(* IEC 61131-3 sources: teller/JD_Teller_LC2_V11/Class/Jamdetection_TeachIn_Teller, 1 file *)

(* ---- Jamdetection_TeachIn_Teller.st ---- *)
(*!
<Class
	Name               = "Jamdetection_TeachIn_Teller"
	Revision           = "1.1"
	RealtimeTask       = "true"
	CyclicTask         = "true"
	BackgroundTask     = "false"
	Sigmatek           = "false"
	OSInterface        = "false"
	HighPriority       = "false"
	Automatic          = "false"
	UpdateMode         = "Prescan"
	SharedCommandTable = "true"
	Objectsize         = "(540,120)">
	<Channels>
		<Server Name="ClassSvr" Visualized="false" Initialize="false" WriteProtected="true" Retentive="false"/>
		<Server Name="CopyTeachIn" Visualized="true" Initialize="false" WriteProtected="false" Retentive="false"/>
		<Server Name="iEncDiv" Visualized="true" Initialize="false" WriteProtected="false" Retentive="false"/>
		<Server Name="iEncMulti" Visualized="true" Initialize="false" WriteProtected="false" Retentive="false"/>
		<Server Name="JamPauze" Visualized="true" Initialize="false" WriteProtected="false" Retentive="false"/>
		<Server Name="MaxLengthBox" Visualized="true" Initialize="false" WriteProtected="false" Retentive="false"/>
		<Server Name="MinJamSpeed" Visualized="true" Initialize="false" WriteProtected="false" Retentive="false"/>
		<Server Name="MinSpot" Visualized="true" Initialize="false" WriteProtected="false" Retentive="false"/>
		<Server Name="Nr_Of_JamSensors" Visualized="true" Initialize="false" WriteProtected="true" Retentive="false"/>
		<Server Name="oJamdetection" Visualized="true" Initialize="false" WriteProtected="true" Retentive="false"/>
		<Server Name="oSpeed" Visualized="true" Initialize="false" WriteProtected="true" Retentive="false"/>
		<Server Name="ResetJam" Visualized="false" Initialize="false" WriteProtected="false" Retentive="false"/>
		<Server Name="Sectie" Visualized="true" Initialize="false" WriteProtected="true" Retentive="false"/>
		<Server Name="SectieNrInMachine" Visualized="true" Initialize="false" WriteProtected="false" Retentive="false"/>
		<Server Name="SectieType" Visualized="true" Initialize="false" WriteProtected="true" Retentive="false"/>
		<Server Name="sExtraBox" Visualized="true" Initialize="false" WriteProtected="false" Retentive="false"/>
		<Server Name="SimSpeed" Visualized="false" Initialize="false" WriteProtected="false" Retentive="false"/>
		<Server Name="Simulator" Visualized="false" Initialize="false" WriteProtected="false" Retentive="false"/>
		<Server Name="TeachIn" Visualized="true" Initialize="false" WriteProtected="false" Retentive="false"/>
		<Client Name="c_JamData" Required="true" Internal="false"/>
		<Client Name="c_SectieType" Required="true" Internal="false"/>
		<Client Name="cJamDetect" Required="false" Internal="false" Comment="Status Jamdetect&#13;&#10;1: Detectie&#13;&#10;0: Geen detectie"/>
		<Client Name="cJamDetect2HW" Required="true" Internal="false"/>
		<Client Name="cJamDetectSignal" Required="false" Internal="false" Comment="Knipperende uitgang"/>
		<Client Name="cJamReset" Required="true" Internal="false"/>
		<Client Name="cSensor_01" Required="false" Internal="false"/>
		<Client Name="cSensor_02" Required="false" Internal="false"/>
		<Client Name="cSensor_03" Required="false" Internal="false"/>
		<Client Name="cSimpuls" Required="false" Internal="false"/>
		<Client Name="iEncoder" Required="false" Internal="false"/>
	</Channels>
	<RevDoku>
		<Owner Company="jd" Author="SV"/>
		<Dokumentation Revision="1.1" Date="2014-09-16" Author="SV" Company="jd" Description="Clients cSensor_4 tm cSensor_16 verwijderd.&#13;&#10;cSimpuls sensoren verwijderd.&#13;&#10;TaskOnOff server verwijderd.&#13;&#10;TaskOnOff uit RT en CY wordk verwijderd."/>
		<Dokumentation Revision="1.0" Date="2014-09-04" Author="SV" Company="jd" Description="Kopie uit retrofit class versie 1.2. De class haalt de neemt nu de EncMul, EncDiv, MinSpot en &#13;&#10;ExtraBox uit de TellerClass_Teller.&#13;&#10;Client Jampauze ingevoerd, regel 244. Zorgt voor tijdelijk negeren van de jamfunctie."/>
	</RevDoku>
</Class>
*)
Jamdetection_TeachIn_Teller : CLASS
	TYPE
#pragma pack(push, 1)
	  tJam : STRUCT
	    Sensor : ARRAY [0..16] OF DINT;
	    CaseMinSSW : ARRAY [0..16] OF DINT;
	    MinimaleCounter : ARRAY [0..16] OF DINT;
	    Din : ARRAY [0..16] OF DINT;
	    JamBoxlength : ARRAY [0..16] OF DINT;
	    JamBoxLengthCalc : ARRAY [0..16] OF DINT;
	    CaseJam : ARRAY [0..16] OF DINT;
	    Jampos : ARRAY [0..16] OF DINT;
	    Jamdetection : ARRAY [0..16] OF DINT;
	    CaseTeachIn : ARRAY [0..16] OF DINT;
	    TeachInLength : ARRAY [0..16] OF DINT;
	    Holes : ARRAY [0..16] OF DINT;
	    Sensor_Aanwezig : ARRAY [0..16] OF DINT;
	    OnOff : ARRAY [0..16] OF DINT;
	  END_STRUCT;
#pragma pack(pop)
	END_TYPE
  //Servers:
	ClassSvr 	: SvrChCmd_DINT;
	Sectie 	: SvrCh_tSectie;
	SectieType 	: SvrCh_DINT;
	Nr_Of_JamSensors 	: SvrCh_DINT;
	SectieNrInMachine 	: SvrCh_DINT;
	MinJamSpeed 	: SvrCh_DINT;
	MinSpot 	: SvrCh_DINT;
	sExtraBox 	: SvrCh_DINT;
	iEncMulti 	: SvrCh_DINT;
	iEncDiv 	: SvrCh_DINT;
	oSpeed 	: SvrCh_DINT;
	SimSpeed 	: SvrCh_DINT;
	Simulator 	: SvrCh_DINT;
	MaxLengthBox 	: SvrCh_DINT;
	oJamdetection 	: SvrCh_DINT;
	ResetJam 	: SvrCh_DINT;
	TeachIn 	: SvrCh_DINT;
	CopyTeachIn 	: SvrCh_DINT;
	JamPauze 	: SvrCh_DINT;
  //Clients:
	c_JamData 	: CltChCmd_RAMex;
	c_SectieType 	: CltCh_DINT;
	iEncoder 	: CltCh_DINT;
	cJamDetect 	: CltCh_DINT;
	cJamDetectSignal 	: CltCh_DINT;
	cJamDetect2HW 	: CltCh_DINT;
	cSensor_01 	: CltCh_DINT;
	cSensor_02 	: CltCh_DINT;
	cSensor_03 	: CltCh_DINT;
	cSimpuls 	: CltCh_DINT;
	cJamReset 	: CltCh_DINT;
  //Variables:
		JamData 	: ^tJamDetect;
		Enc 	: Encoder1;
		Jam 	: tJam;
		OSpeedie 	: tOspeed;
		i 	: DINT;
		ii 	: DINT;
		iii 	: DINT;
		Reset 	: DINT;
		Teach 	: DINT;
		Timer 	: UDINT;
		Timer2 	: UDINT;
		Timer3 	: UDINT;
		caseKnipper 	: DINT;
		cJamDetectSignalOld 	: DINT;
		caseJam2HW 	: DINT;
		JamDetPrevState 	: DINT;
  //Functions:

	FUNCTION VIRTUAL GLOBAL Init;

	FUNCTION VIRTUAL GLOBAL CyWork
		VAR_INPUT
			EAX 	: UDINT;
		END_VAR
		VAR_OUTPUT
			state (EAX) 	: UDINT;
		END_VAR;

	FUNCTION VIRTUAL GLOBAL RtWork
		VAR_INPUT
			EAX 	: UDINT;
		END_VAR
		VAR_OUTPUT
			state (EAX) 	: UDINT;
		END_VAR;

	FUNCTION VIRTUAL GLOBAL Nr_Of_JamSensors::Write
		VAR_INPUT
			input (EAX) 	: DINT;
		END_VAR
		VAR_OUTPUT
			result (EAX) 	: DINT;
		END_VAR;

	FUNCTION VIRTUAL GLOBAL SectieNrInMachine::Write
		VAR_INPUT
			input (EAX) 	: DINT;
		END_VAR
		VAR_OUTPUT
			result (EAX) 	: DINT;
		END_VAR;

	FUNCTION VIRTUAL GLOBAL MinJamSpeed::Write
		VAR_INPUT
			input (EAX) 	: DINT;
		END_VAR
		VAR_OUTPUT
			result (EAX) 	: DINT;
		END_VAR;

	FUNCTION VIRTUAL GLOBAL MinSpot::Write
		VAR_INPUT
			input (EAX) 	: DINT;
		END_VAR
		VAR_OUTPUT
			result (EAX) 	: DINT;
		END_VAR;

	FUNCTION VIRTUAL GLOBAL sExtraBox::Write
		VAR_INPUT
			input (EAX) 	: DINT;
		END_VAR
		VAR_OUTPUT
			result (EAX) 	: DINT;
		END_VAR;

	FUNCTION VIRTUAL GLOBAL iEncMulti::Write
		VAR_INPUT
			input (EAX) 	: DINT;
		END_VAR
		VAR_OUTPUT
			result (EAX) 	: DINT;
		END_VAR;

	FUNCTION VIRTUAL GLOBAL iEncDiv::Write
		VAR_INPUT
			input (EAX) 	: DINT;
		END_VAR
		VAR_OUTPUT
			result (EAX) 	: DINT;
		END_VAR;

	FUNCTION VIRTUAL GLOBAL MaxLengthBox::Write
		VAR_INPUT
			input (EAX) 	: DINT;
		END_VAR
		VAR_OUTPUT
			result (EAX) 	: DINT;
		END_VAR;

	FUNCTION VIRTUAL GLOBAL ResetJam::Write
		VAR_INPUT
			input (EAX) 	: DINT;
		END_VAR
		VAR_OUTPUT
			result (EAX) 	: DINT;
		END_VAR;

	FUNCTION VIRTUAL GLOBAL TeachIn::Write
		VAR_INPUT
			input (EAX) 	: DINT;
		END_VAR
		VAR_OUTPUT
			result (EAX) 	: DINT;
		END_VAR;

	FUNCTION VIRTUAL GLOBAL CopyTeachIn::Write
		VAR_INPUT
			input (EAX) 	: DINT;
		END_VAR
		VAR_OUTPUT
			result (EAX) 	: DINT;
		END_VAR;
  //Tables:
	FUNCTION @STD
		VAR_OUTPUT
			ret_code	: CONFSTATES;
		END_VAR;
	FUNCTION GLOBAL TAB @CT_;
END_CLASS;

#pragma usingLtd RAMex

FUNCTION VIRTUAL GLOBAL Jamdetection_TeachIn_Teller::Init
VAR
	ii: DINT;
END_VAR

  if      c_JamData.GetSize() <> sizeof(tJamDetect) then
          c_JamData.SetSize(udSize:=sizeof(tJamDetect));
  end_if;

  if      _FirstScan then
          JamData := (c_JamData.GetDataPtr())$^tJamDetect;
          SectieType := c_SectieType;
          if    SectieType < 1 then
                SectieType := 1;
          elsif SectieType > 12 then
                SectieType := 12;
          end_if;

          if    SectieType = 1 then
                Sectie := PreFeeder;
          elsif SectieType = 2 then
                Sectie := TriFeeder;
          elsif SectieType = 3 then
                Sectie := Feeder;
          elsif SectieType = 4 then
                Sectie := MAS;
          elsif SectieType = 5 then
                Sectie := Prefold;
          elsif SectieType = 6 then
                Sectie := A_Sectie;
          elsif SectieType = 7 then
                Sectie := B_Sectie;
          elsif SectieType = 8 then
                Sectie := C_Sectie;
          elsif SectieType = 9 then
                Sectie := FinalFold;
          elsif SectieType = 10 then
                Sectie := F_Unit;
          elsif SectieType = 11 then
                Sectie := Trombone;
          elsif SectieType = 12 then
                Sectie := ConveyorBand;
          end_if;

          Nr_Of_JamSensors.Write(input:=JamData^.NrOfJamSensors);
          MinSpot.Write(input:=JamData^.MinSpot);
          sExtraBox.Write(input:=JamData^.sExtraBox);
          iEncMulti.Write(input:=JamData^.iEncMulti);
          iEncDiv.Write(input:=JamData^.iEncDiv);
          MaxLengthBox.Write(input:=JamData^.T_Doos);
          MinJamSpeed.Write(input:=JamData^.MinJamSpeed);
          SectieNrInMachine.Write(input:=JamData^.SectieNrInMachine);
          //SV max aantal sensoren
          Nr_Of_JamSensors := 3;
          for ii:= Nr_Of_JamSensors to 16 do
              JamData^.Status[ii] := No_Sensor_Configurated;
          end_for;

          JamData^.NrOfJamSensors := Nr_Of_JamSensors;
  end_if;

END_FUNCTION

FUNCTION VIRTUAL GLOBAL Jamdetection_TeachIn_Teller::RtWork
	VAR_INPUT
		EAX 	: UDINT;
	END_VAR
	VAR_OUTPUT
		state (EAX) 	: UDINT;
	END_VAR

//Als in de machine setup de functie is geselelecteerd wordt de code uitgevoerd

      if  Nr_Of_JamSensors > 0 then

      //inlezen van de encoder

        if    SimSpeed <= 0 then
              iEncoder := iEncoder.Read();
        else
              iEncoder += SimSpeed;
        end_if;

        if    enc.Divider < 1 then
              enc.Divider := 1;
        end_if;

        Enc.EncoderDelta := iEncoder - Enc.EncoderOld;
        Enc.EncoderOld := iEncoder;
        Enc.SpeedDelta := ((Enc.EncoderDelta * encres * enc.Multi) / enc.Divider);

        if  ResetJam then
            Reset := 1;
            ResetJam := 0;
        end_if;

        for i:= 1 to Nr_Of_JamSensors do

          if Simulator = 0 then //Simulator puls aan of uit
            //Sensoren inlezen
            if    i = 1 then
                  cSensor_01 := cSensor_01.Read();
                  Jam.Sensor[1] := cSensor_01;
            elsif i = 2 then
                  cSensor_02 := cSensor_02.Read();
                  Jam.Sensor[2] := cSensor_02;
            elsif i = 3 then
                  cSensor_03 := cSensor_03.Read();
                  Jam.Sensor[3] := cSensor_03;

            end_if;
          else //simulator puls          SV 16-09-2014 sensoren 4 tm 16 verwijderd
            cSimpuls := cSimpuls.Read();
            Jam.Sensor[1] := cSimpuls;
            Jam.Sensor[2] := cSimpuls;
            Jam.Sensor[3] := cSimpuls;

                                      // SV 16-09-2014 sensoren 4 tm 16 verwijderd
            cSensor_01 :=  Jam.Sensor[1];
            cSensor_02 :=  Jam.Sensor[2];
            cSensor_03 :=  Jam.Sensor[3];

          end_if;

            //Minspot
                case Jam.CaseMinSSW[i] of
                0:
                  if  Jam.Sensor[i] = 1 then
                      Jam.MinimaleCounter[i]:=0;
                      Jam.Din[i]:=0;
                      Jam.CaseMinSSW[i]+=1;
                  end_if;
                1:
                  Jam.MinimaleCounter[i]+= Enc.SpeedDelta;

                  if  Jam.MinimaleCounter[i] > (MinSpot * encres) then
                      if  Jam.Sensor[i] = 1 then
                          Jam.Din[i]:=1;
                          Jam.CaseMinSSW[i]+=1;
                      else
                          Jam.CaseMinSSW[i]:=0;
                      end_if;
                  end_if;
                2:
                      Jam.Din[i]:=0;
                  if  Jam.Sensor[i] = 0 then
                      Jam.CaseMinSSW[i]:=0;
                  end_if;
                end_case;

            //Jam
                if Jam.JamBoxlength[i] <> 0 & Teach = 0  & Jam.OnOff[i]  then
                    case Jam.CaseJam[i] of
                    0: //controleren of aan de snipper beveiliging is voldaan
                       if Jam.Din[i] then
                          Jam.CaseJam[i] += 1;
                          Jam.Jampos[i] :=  MinSpot * encres;
                          Jam.JamBoxLengthCalc[i] := (Jam.JamBoxlength[i] + sExtraBox) * encres;
                       end_if;
                    1: //Controle op Jamdetect
                       //Kijken of de sensor hoog is na de ingestelde Boxlengte en extra waarde
                       //Onder een bepaalde snelheid wordt de jamdetect niet aangestuurd
                          Jam.Jampos[i] += Enc.SpeedDelta;
                          if   Jam.Jampos[i] > Jam.JamBoxLengthCalc[i] then //De Jampos loopt nu mee
                              if   Jam.Sensor[i] & (MinJamSpeed < oSpeed) & (JamPauze = 0) then     //2014-09-04 SV Cient JamPauze ingevoerd.
                                   Jam.Jamdetection[i] := 1;
                                   oJamdetection := 1;
                                   Jam.CaseJam[i] += 1;
                              else                                //Geen Jamdetect!!
                                   Jam.Jamdetection[i] := 0;      //Geen Jamdetect, terug naar stap 0 en wachten op een nieuwe doos
                                   Jam.CaseJam[i] := 0;
                              end_if;
                          end_if;
                    2:  //Jam, reset is nodig om verder te gaan.

                       if Reset then
                          Jam.Jamdetection[i] := 0;
                          oJamdetection := 0;
                          //als bij reset de doos niet is weggehaald start de controle opnieuw
                          //if  Jam.Sensor[i] = 1 then
                              //Jam.CaseJam[i] := 1;
                              //Jam.Jampos[i] :=  MinSpot * encres;
                              //Jam.JamBoxLengthCalc[i] := (Jam.JamBoxlength[i] + sExtraBox) * encres;
                          //else
                              Jam.CaseJam[i]:=0;

                          //end_if;
                       end_if;
                     end_case;

                 end_if;

              //TeachIn
              //Holes kunnen worden gezien

              if Teach = 1  then
                  case Jam.CaseTeachIn[i] of
                  0:
                       if     Jam.Din[i] then
                              Jam.CaseTeachIn[i] += 1;
                              Jam.Jampos[i] :=  MinSpot * encres;
                       end_if;
                  1:
                       Jam.Jampos[i] += Enc.SpeedDelta;

                       //Bij geblokkeerde sensor error aangeven
                       if     jam.Sensor[i] = 1 & Jam.Jampos[i] >= ((MaxLengthBox + sExtraBox) * encres) then
                              Jam.TeachInLength[i] := 0;
                              JamData^.Status[i] := Box_Oversized;
                              Jam.CaseTeachIn[i] := 3;
                       //Box detected save position
                       elsif  jam.Sensor[i] = 0  then
                              Jam.TeachInLength[i] := Jam.Jampos[i];
                              Jam.CaseTeachIn[i] += 1;
                       end_if;

                  2:
                       Jam.Jampos[i] += Enc.SpeedDelta;

                       //Er is een gat gedetecteerd Hole
                       if     jam.Sensor[i] = 1 & Jam.Jampos[i] < ((MaxLengthBox + sExtraBox) * encres) then
                              Jam.Holes[i] += 1;
                              Jam.CaseTeachIn[i] := 1;
                       //Ready
                       elsif  jam.Sensor[i] = 0 & Jam.Jampos[i] >= ((MaxLengthBox + sExtraBox) * encres) then
                              if    jam.holes[i] > 0 then
                                    JamData^.Status[i] := Holes_Detected;
                              else
                                    JamData^.Status[i] := TeachIn_Ok;
                              end_if;
                              Jam.CaseTeachIn[i] := 3;
                       elsif  jam.Sensor[i] = 1 & Jam.Jampos[i] >= ((MaxLengthBox + sExtraBox) * encres) then
                              Jam.TeachInLength[i] := 0;
                              JamData^.Status[i] := Box_Oversized;
                              Jam.CaseTeachIn[i] := 3;
                       end_if;

                  3:   //Ready
                       //Do nothing

                  end_case;

              end_if;
        end_for;

        Reset := 0;
      end_if;

	state := READY;

END_FUNCTION

FUNCTION VIRTUAL GLOBAL Jamdetection_TeachIn_Teller::CyWork
	VAR_INPUT
		EAX 	: UDINT;
	END_VAR
	VAR_OUTPUT
		state (EAX) 	: UDINT;
	END_VAR

//Als in de machine setup de functie is geselelecteerd wordt de code uitgevoerd

      if  Nr_Of_JamSensors > 0 then

        //encoder

        if iEncDiv = 0 then
           iEncDiv :=1;
        end_if;

        if    SimSpeed <= 0 then
              Enc.Multi   := iEncMulti;
              Enc.Divider := iEncDiv;

              OSpeedie.EncIn :=iEncoder;
              ospeedie.EncDelta := OSpeedie.EncIn - OSpeedie.EncOud;
              OSpeedie.EncOud := OSpeedie.EncIn;
              oSpeed := to_dint((to_Real(ospeedie.EncDelta) * 60 * To_Real(Enc.Multi)) / (to_Real(Enc.Divider)*50));
        else
              Enc.Multi   := 1000;
              Enc.Divider := 60000;
              oSpeed := SimSpeed;
        end_if;

        for ii:= 1 to Nr_Of_JamSensors do
            Jam.JamBoxlength[ii] := JamData^.JamBoxlength[ii];
            Jam.OnOff[ii] := JamData^.OnOff[ii];
            JamData^.TeachInLength[ii] := jam.TeachInLength[ii];

            if  Jam.Jamdetection[ii] = 1 then
                JamData^.Status[ii] := Jam_Detect;
            end_if;

            if  Teach = 0 & (Jam.JamBoxlength[ii] = 0 | Jam.OnOff[ii] = 0)  then
                JamData^.Status[ii] := Turned_Off;
            end_if;

            JamData^.TeachInLength[ii] := Jam.TeachInLength[ii]/encres;

            JamData^.Sensor[ii] := Jam.Sensor[ii];

        end_for;

        cJamDetect := oJamdetection;
        cJamDetect.Write(input:=cJamDetect);

        if     oJamdetection = 1 then
               //noodstop bedienen
               if     caseJam2HW = 0 then
                      caseJam2HW := 1;
               end_if;

               case   caseKnipper of

               0:
                      timer := ops.tAbsolute;
                      cJamDetectSignal := 1;
                      caseKnipper := 1;

               1:
                      if  ops.tAbsolute - timer > 125 then
                          timer := ops.tAbsolute;
                          caseKnipper := 2;
                      end_if;

               2:
                      timer := ops.tAbsolute;
                      cJamDetectSignal := 0;
                      caseKnipper := 3;

               3:
                      if  ops.tAbsolute - timer > 125 then
                          timer := ops.tAbsolute;
                          caseKnipper := 0;
                      end_if;
               end_case;

        else
               caseKnipper := 0;
               cJamDetectSignal := 0;

               //noodstop uitsturing moet cyclus afgerond hebben!
               if   caseJam2HW = 3 then
                    caseJam2HW := 0;
               end_if;

        end_if;

        //stopcircuit 1 seconde onderbreken
        case   caseJam2HW   of

        0:     //Doe niets

        1:
               cJamDetect2HW := 1;
               cJamDetect2HW.Write(input:=cJamDetect2HW);
               caseJam2HW += 1;
               Timer3 := ops.tAbsolute;

        2:
               //HW uitschakelen
               if    ops.tAbsolute - Timer3 > 1000 then
                     cJamDetect2HW := 0;
                     cJamDetect2HW.Write(input:=cJamDetect2HW);
                     caseJam2HW += 1;
               end_if;

        3:     //doe niets

        end_case;

        if     cJamDetectSignalOld <> cJamDetectSignal  then
               cJamDetectSignalOld := cJamDetectSignal;
               cJamDetectSignal.Write(input:=cJamDetectSignal);

        end_if;

      end_if;

  //SV 29-8-2014. Instellinen die dezelfde waarde hebben als de TellerClass overnemen uit de TellerClass,  zodat dit maar 1 keer hoeft te worden ingegeven..
  MinSpot := JamData^.MinSpot;
  sExtraBox := JamData^.sExtraBox;
  iEncMulti := JamData^.iEncMulti;
  iEncDiv := JamData^.iEncDiv;

	state := READY;

END_FUNCTION

FUNCTION VIRTUAL GLOBAL Jamdetection_TeachIn_Teller::Nr_Of_JamSensors::Write
	VAR_INPUT
		input (EAX) 	: DINT;
	END_VAR
	VAR_OUTPUT
		result (EAX) 	: DINT;
	END_VAR

	Nr_Of_JamSensors := input;
  if  Nr_Of_JamSensors < 0 | Nr_Of_JamSensors > 16 then
      Nr_Of_JamSensors := 0;
  end_if;

  for ii:= Nr_Of_JamSensors to 16 do
      JamData^.Status[ii] := No_Sensor_Configurated;
  end_for;

  JamData^.NrOfJamSensors := Nr_Of_JamSensors;

 	result := Nr_Of_JamSensors;

END_FUNCTION

FUNCTION VIRTUAL GLOBAL Jamdetection_TeachIn_Teller::MinSpot::Write
	VAR_INPUT
		input (EAX) 	: DINT;
	END_VAR
	VAR_OUTPUT
		result (EAX) 	: DINT;
	END_VAR

	MinSpot := input;
  if    MinSpot < 20 then
        MinSpot := 20;
  elsif MinSpot > 100 then
        MinSpot := 20;
  end_if;

  JamData^.MinSpot := MinSpot;

 	result := MinSpot;

END_FUNCTION

FUNCTION VIRTUAL GLOBAL Jamdetection_TeachIn_Teller::sExtraBox::Write
	VAR_INPUT
		input (EAX) 	: DINT;
	END_VAR
	VAR_OUTPUT
		result (EAX) 	: DINT;
	END_VAR

	sExtraBox := input;
  if    sExtraBox < 20 then
        sExtraBox := 20;
  elsif sExtraBox > 100 then
        sExtraBox := 20;
  end_if;
  JamData^.sExtraBox := sExtraBox;

 	result := sExtraBox;

END_FUNCTION

FUNCTION VIRTUAL GLOBAL Jamdetection_TeachIn_Teller::iEncMulti::Write
	VAR_INPUT
		input (EAX) 	: DINT;
	END_VAR
	VAR_OUTPUT
		result (EAX) 	: DINT;
	END_VAR

	iEncMulti := input;
  JamData^.iEncMulti := iEncMulti;

 	result := iEncMulti;

END_FUNCTION

FUNCTION VIRTUAL GLOBAL Jamdetection_TeachIn_Teller::iEncDiv::Write
	VAR_INPUT
		input (EAX) 	: DINT;
	END_VAR
	VAR_OUTPUT
		result (EAX) 	: DINT;
	END_VAR

	iEncDiv := input;
  if iEncDiv < 1 then
     iEncDiv := 1;
  end_if;

  JamData^.iEncDiv := iEncDiv;
 	result := iEncDiv;

END_FUNCTION

FUNCTION VIRTUAL GLOBAL Jamdetection_TeachIn_Teller::MaxLengthBox::Write
	VAR_INPUT
		input (EAX) 	: DINT;
	END_VAR
	VAR_OUTPUT
		result (EAX) 	: DINT;
	END_VAR

	MaxLengthBox := input;
  if    MaxLengthBox < 2000 then
        MaxLengthBox := 2000;
  elsif MaxLengthBox > 5000 then
        MaxLengthBox := 5000;
  end_if;
  JamData^.T_Doos := MaxLengthBox;

 	result := MaxLengthBox;

END_FUNCTION

FUNCTION VIRTUAL GLOBAL Jamdetection_TeachIn_Teller::MinJamSpeed::Write
	VAR_INPUT
		input (EAX) 	: DINT;
	END_VAR
	VAR_OUTPUT
		result (EAX) 	: DINT;
	END_VAR

	MinJamSpeed := input;
  if    MinJamSpeed < 0 | MinJamSpeed > 250  then
        MinJamSpeed := 0;
  end_if;
  JamData^.MinJamSpeed := MinJamSpeed;

 	result := MinJamSpeed;

END_FUNCTION

FUNCTION VIRTUAL GLOBAL Jamdetection_TeachIn_Teller::ResetJam::Write
	VAR_INPUT
		input (EAX) 	: DINT;
	END_VAR
	VAR_OUTPUT
		result (EAX) 	: DINT;
	END_VAR

	ResetJam := input;

  if  ResetJam < 0 | ResetJam > 1 then
      ResetJam := 0;
  end_if;

  for ii:= 1 to Nr_Of_JamSensors do
     if JamData^.Status[ii] = Jam_Detect then
        JamData^.Status[ii] := Normal_Operation;
     end_if;
  end_for;

 	result := ResetJam;

END_FUNCTION

FUNCTION VIRTUAL GLOBAL Jamdetection_TeachIn_Teller::TeachIn::Write
	VAR_INPUT
		input (EAX) 	: DINT;
	END_VAR
	VAR_OUTPUT
		result (EAX) 	: DINT;
	END_VAR

	TeachIn := input;

  //Zonder T waarde doos geen TeachIn!!!
  if    MaxLengthBox = 0 | TeachIn = 0 then
        Teach := 0;

        //Teach in case resettem
        for   iii := 1 to Nr_Of_JamSensors do
              Jam.CaseTeachIn[iii] := 0;
              jam.Holes[iii] := 0;
              Jam.TeachInLength[iii] := 0;
              if JamData^.OnOff[iii] > 0 & JamData^.JamBoxlength[iii] > 0 then
                 JamData^.Status[iii] := Normal_Operation;
              end_if;
        end_for;

  else
        Teach := 1;
        TeachIn := 1;

        //Reset eventuele eerdere jamdetect
        oJamdetection := 0;

        for   iii := 1 to Nr_Of_JamSensors do
              Jam.Jamdetection[iii] := 0;
              Jam.CaseJam[iii]:=0;

              //Start status
              JamData^.Status[iii] := No_Box_Detected;

              Jam.CaseTeachIn[iii] := 0;
              jam.Holes[iii] := 0;
              Jam.TeachInLength[iii] := 0;

        end_for;
  end_if;

 	result := TeachIn;

END_FUNCTION

FUNCTION VIRTUAL GLOBAL Jamdetection_TeachIn_Teller::CopyTeachIn::Write
	VAR_INPUT
		input (EAX) 	: DINT;
	END_VAR
	VAR_OUTPUT
		result (EAX) 	: DINT;
	END_VAR

	CopyTeachIn := input;

  CopyTeachIn := 0;
  TeachIn := 0;
  Teach := 0;

  for   iii := 1 to Nr_Of_JamSensors do
        JamData^.JamBoxlength[iii] := Jam.TeachInLength[iii]/ encres;
        if    JamData^.TeachInLength[iii] > 0 then
              JamData^.Status[iii] := Normal_Operation;
        else
              JamData^.Status[iii] := Turned_Off;
        end_if;
  end_for;

 	result := CopyTeachIn;

END_FUNCTION

FUNCTION VIRTUAL GLOBAL Jamdetection_TeachIn_Teller::SectieNrInMachine::Write
	VAR_INPUT
		input (EAX) 	: DINT;
	END_VAR
	VAR_OUTPUT
		result (EAX) 	: DINT;
	END_VAR

	SectieNrInMachine := input;
  if SectieNrInMachine < 0 then
     SectieNrInMachine := 0;
  end_if;
  if SectieNrInMachine > 18 then
     SectieNrInMachine :=18;
  end_if;

  JamData^.SectieNrInMachine := SectieNrInMachine;

 	result := SectieNrInMachine;

END_FUNCTION
